FUNCTION_BLOCK FB_HE_SATT_FilterCombination IMPLEMENTS I_HE_SATT_FilterCombination
VAR
    aiFilter : ARRAY[1..PL_HE_SATT_Parameters.nNumHolders] OF I_HE_SATT_Filter;
    nHolderNumberOfLastFilterAdded : INT;
END_VAR


METHOD AddFilter
VAR_INPUT
	nHolderNumber	: INT;
	iFilter	: I_HE_SATT_Filter;
END_VAR

IF NOT THIS^.IsValidHolderNumber(nHolderNumber := nHolderNumber) THEN
    RETURN;
END_IF

THIS^.aiFilter[nHolderNumber] := iFilter;

THIS^.nHolderNumberOfLastFilterAdded := nHolderNumber;
END_METHOD


METHOD Clear
VAR
    nIteratorHolder : INT;
END_VAR

FOR nIteratorHolder := 1 TO PL_HE_SATT_Parameters.nNumHolders BY 1 DO
    aiFilter[nIteratorHolder] := 0;
END_FOR
END_METHOD


METHOD GetFilter : I_HE_SATT_Filter
VAR_INPUT
    nHolderNumber : INT;
END_VAR

GetFilter := THIS^.aiFilter[nHolderNumber];
END_METHOD


PROPERTY HolderNumberOfLastFilterAdded : INT
GET

HolderNumberOfLastFilterAdded := THIS^.nHolderNumberOfLastFilterAdded;
END_GET
END_PROPERTY


METHOD PUBLIC IsValidHolderNumber : BOOL
VAR_INPUT
    nHolderNumber : INT;
END_VAR

IF nHolderNumber >= 1 AND nHolderNumber <= PL_HE_SATT_Parameters.nNumHolders THEN
    IsValidHolderNumber := TRUE;
END_IF
END_METHOD


METHOD RemoveFilter
VAR_INPUT
	nHolderNumber	: INT;
END_VAR

IF NOT THIS^.IsValidHolderNumber(nHolderNumber := nHolderNumber) THEN
    RETURN;
END_IF

THIS^.aiFilter[nHolderNumber] := 0;
END_METHOD

END_FUNCTION_BLOCK

(* stored: Version 1.1.0.1
   POU FB_HE_SATT_FilterCombination: Id {3f5c161d-1dfa-48b6-b045-ee3172059675}, SpecialFunc None
   Method AddFilter: Id {49246903-5cd5-45d9-b201-71e59c896238}
   Method Clear: Id {fc41e55f-411e-43c9-bca4-e1a17785476b}
   Method GetFilter: Id {8f99526e-89c4-4076-a4d2-8f5516465bd6}
   Property HolderNumberOfLastFilterAdded: Id {2725ac41-65d3-46b9-87a3-6477d388d25f}
   Get Get: Id {171c8033-4a4d-4327-8d62-5b55a130569b}
   Method IsValidHolderNumber: Id {72e9bbce-8dd2-449c-a056-f356a1b70094}
   Method RemoveFilter: Id {e4fa1af3-e2be-41a6-8f51-e9bee6544b1f} *)
